PROGRAM Ax_01_AxisMoveTypeSelect_02
VAR
	HMI_Motion: FB_HMI_Control;


	tMessageOffset: UINT;
	tNumMessagesPerRow: UINT;
	
	
	MyAdvanceInterlock: BOOL;
	MyReturnInterlock: BOOL;
	
	MyAutoAdvanceCondition: BOOL;
	MyAutoReturnCondition: BOOL;
	
	myAdvancePrompt: BOOL;
	myReturnPrompt: BOOL;
	

	NotUsed: UINT;
END_VAR

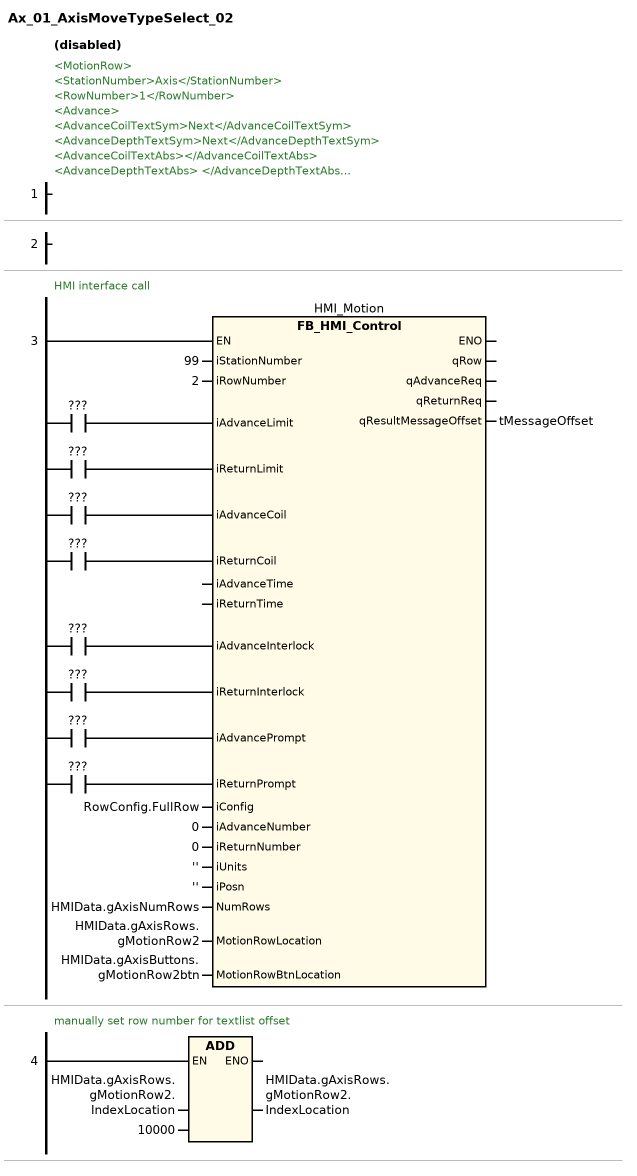
// NETWORK 1 (disabled)
// <MotionRow>
// <StationNumber>Axis</StationNumber>
// <RowNumber>1</RowNumber>
//   <Advance>
//     <AdvanceCoilTextSym>Next</AdvanceCoilTextSym>
//     <AdvanceDepthTextSym>Next</AdvanceDepthTextSym>
//     <AdvanceCoilTextAbs></AdvanceCoilTextAbs>
//     <AdvanceDepthTextAbs> </AdvanceDepthTextAbs>
//     <ManSeq></ManSeq>
//   </Advance>
//   <Return>
//     <ReturnCoilTextSym>Previous</ReturnCoilTextSym>
//     <ReturnDepthTextSym>Previous</ReturnDepthTextSym>
//     <ReturnCoilTextAbs></ReturnCoilTextAbs>
//     <ReturnDepthTextAbs></ReturnDepthTextAbs>
//    <ManSeq></ManSeq>
//   </Return>
//   <Motion>
//     <NameSym>Axis Name</NameSym>
//     <NameAbs>X1</NameAbs>
//   </Motion>
// </MotionRow>

// NETWORK 2

// NETWORK 3
// HMI interface call
HMI_Motion(
    iStationNumber := 99,
    iRowNumber := 2,
    iConfig := RowConfig.FullRow,
    iAdvanceNumber := 0,
    iReturnNumber := 0,
    iUnits := '',
    iPosn := '',
    NumRows := HMIData.gAxisNumRows,
    MotionRowLocation := HMIData.gAxisRows.gMotionRow2,
    MotionRowBtnLocation := HMIData.gAxisButtons.gMotionRow2btn,
    qResultMessageOffset => tMessageOffset); // FB_HMI_Control

// NETWORK 4
// manually set row number for textlist offset
HMIData.gAxisRows.gMotionRow2.IndexLocation := HMIData.gAxisRows.gMotionRow2.IndexLocation + 10000;

END_PROGRAM

(* stored: Version 1.1.0.1, ProductVersion 3.1.4024.12
   POU Ax_01_AxisMoveTypeSelect_02: Id {193668af-76f6-42c2-8f7d-eb8927314956}, SpecialFunc None *)
